% RSLogix 500 project BAW TYK 4_BAK001.RSS, saved by version 8.40.00.08 %
PROJECT "UNTITLED"    % processor: type code 33 %

PROGRAM FILES
  LAD 2   11 rungs

DATA FILES
  S2 STATUS  164 elements
  B3 BINARY  1 elements
  T4 TIMER  1 elements
  C5 COUNTER  1 elements
  R6 CONTROL  1 elements
  N7 INTEGER  1 elements
  F8 FLOAT  1 elements

LADDER 2
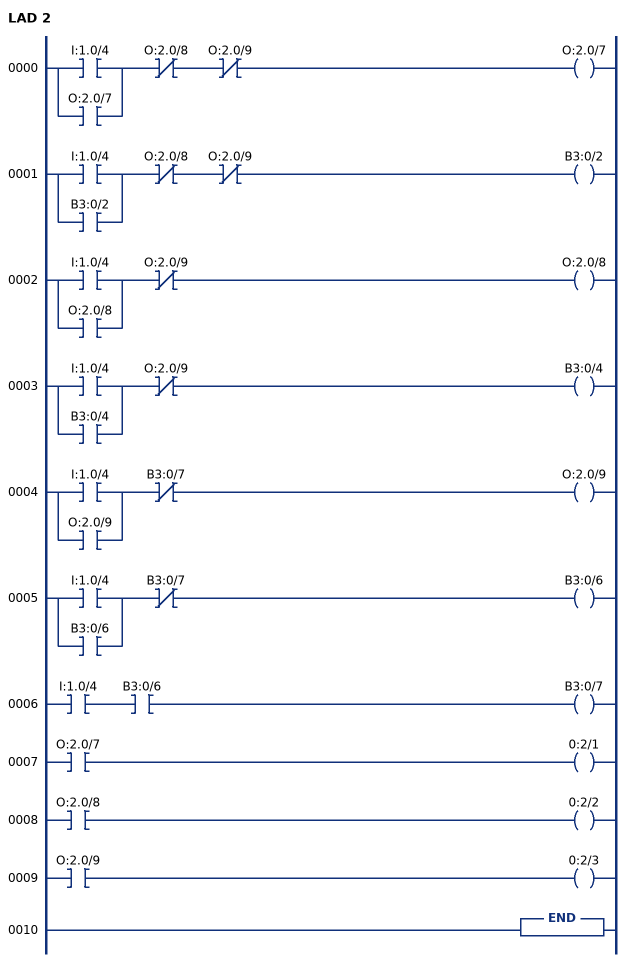
% Rung: 0 %  % edit flag set %
SOR BST XIC I:1.0/4 NXB XIC O:2.0/7 BND XIO O:2.0/8 XIO O:2.0/9 OTE O:2.0/7 EOR
% Rung: 1 %  % edit flag set %
SOR BST XIC I:1.0/4 NXB XIC B3:0/2 BND XIO O:2.0/8 XIO O:2.0/9 OTE B3:0/2 EOR
% Rung: 2 %  % edit flag set %
SOR BST XIC I:1.0/4 NXB XIC O:2.0/8 BND XIO O:2.0/9 OTE O:2.0/8 EOR
% Rung: 3 %  % edit flag set %
SOR BST XIC I:1.0/4 NXB XIC B3:0/4 BND XIO O:2.0/9 OTE B3:0/4 EOR
% Rung: 4 %  % edit flag set %
SOR BST XIC I:1.0/4 NXB XIC O:2.0/9 BND XIO B3:0/7 OTE O:2.0/9 EOR
% Rung: 5 %  % edit flag set %
SOR BST XIC I:1.0/4 NXB XIC B3:0/6 BND XIO B3:0/7 OTE B3:0/6 EOR
% Rung: 6 %  % edit flag set %
SOR XIC I:1.0/4 XIC B3:0/6 OTE B3:0/7 EOR
% Rung: 7 %  % edit flag set %
SOR XIC O:2.0/7 OTE 0:2/1 EOR
% Rung: 8 %  % edit flag set %
SOR XIC O:2.0/8 OTE 0:2/2 EOR
% Rung: 9 %  % edit flag set %
SOR XIC O:2.0/9 OTE 0:2/3 EOR
% Rung: 10 %
SOR END EOR
